// TIA Portal V21 export
TYPE "ST_Button"
   STRUCT
      start : Bool;
      stop : Bool;
      reset : Bool;
      emergencyStop : Bool;
      suspendResume : Bool;
      manualMode : Bool;
      manualRed : Bool;
      manualYellow : Bool;
      manualGreen : Bool;
      pedestrian : Bool;
   END_STRUCT;
END_TYPE
